(* Logix 5000 project; controller Comas_L4 vendor 1 type 14 code 193 rev 30.11; software revision 30.02; part 9 of 12 *)
(* tags used below, declared in another part *)
   Activation_Mode_Once : BOOL;
   Activation_Pompe : BOOL;
   Activation_Synchro_Directe_Codeur : BOOL;
   AOI_Pilotage_Codeur_Vitesse_Moy : Pilotage_Vitesse_Rapide_V4;
   Axe_Comas : MOTION_GROUP;
   Axe_Coupe_Fil : AXIS_CIP_DRIVE;
   Axe_Horizontal_Droit : AXIS_CIP_DRIVE;
   Axe_Horizontal_Gauche : AXIS_CIP_DRIVE;
   Axe_Pompe_Doseuse : AXIS_CIP_DRIVE;
   Axe_Vertical_Droit : AXIS_CIP_DRIVE;
   Axe_Vertical_Gauche : AXIS_CIP_DRIVE;
   Axe_Virtuel_Codeur : AXIS_VIRTUAL;
   Axe_Virtuel_Maitre : AXIS_VIRTUAL;
   CAM_Inter_Virtuel_Maitre : CAM[100];
   CamGenerator_Horizontal : AOI_CamGenerator_ST;
   CamGenerator_Vertical : AOI_CamGenerator_ST;
   CO_Acquit_defaut : BOOL;
   CO_Activation : BOOL;
   CO_Axe_Reel_Desynchro : BOOL;
   CO_Axe_Reel_En_Synchro : BOOL;
   CO_Consigne_Pompe_Acc_Dec : REAL;
   CO_Consigne_Pompe_Jerk : REAL;
   CO_Control_Pompe_Vitesse : REAL;
   CO_Degagement_En_Cours : BOOL;
   CO_Degagement_Possible : BOOL;
   CO_demande_darret : BOOL;
   CO_Demande_Init : BOOL;
   CO_en_Marche : BOOL;
   CO_Engage_Axe_Coupe_Fil : Engage_Axe;
   CO_Engage_Axe_H_Droit : Engage_Axe;
   CO_Engage_Axe_H_Gauche : Engage_Axe;
   CO_Engage_Axe_V_Droit : Engage_Axe;
   CO_Engage_Axe_V_Gauche : Engage_Axe;
   CO_Engage_Maitre : Engage_Axe_Virtuel;
   CO_Engagement : BOOL;
   CO_Engagement_Maitre : BOOL;
   CO_Front_Demande_Init : BOOL;
   CO_Front_Raz_Init : BOOL;
   CO_Front_Reset_Init_OK : BOOL;
   CO_Init_Coupe_Fil : BOOL;
   CO_Init_Horizontal_Droit : BOOL;
   CO_Init_Horizontal_Gauche : BOOL;
   CO_Init_Ok : BOOL;
   CO_Init_Pompe_Doseuse : BOOL;
   CO_Init_Vertical_Droit : BOOL;
   CO_Init_Vertical_Gauche : BOOL;
   CO_Machine_sans_defaut : BOOL;
   CO_Synchro_Axe_En_Cours : BOOL;
   CO_Temp_Activation : TIMER;
   CO_Temp_Desynchro : TIMER;
   CO_Temp_Pret : TIMER;
   CO_Tempo_Demande_Init : TIMER;
   CO_Tempo_Engagement : TIMER;
   CO_TON_Activation : TIMER;
   CO_Top_Degagement : BOOL;
   CO_Top_Depart_Pompe_Avance : BOOL;
   CO_Top_Depart_Pompe_Inter1 : BOOL;
   CO_Top_Depart_Pompe_Inter2 : BOOL;
   CO_Top_Depart_Pompe_Inter3 : BOOL;
   CO_Top_Depart_Pompe_Inter4 : BOOL;
   CO_Top_Depart_Pompe_Inter5 : BOOL;
   CO_Top_Depart_Pompe_Inter6 : BOOL;
   CO_Top_Depart_Pompe_Inter7 : BOOL;
   CO_Top_Depart_Pompe_Inter8 : BOOL;
   CO_Top_Depart_Pompe_Recul : BOOL;
   CO_Top_Once_Axe_Virtuel : BOOL;
   Init_Coupe_Fil : Init_Axe_CIP;
   Init_Horizontal_Droit : Init_Axe_CIP;
   Init_Horizontal_Gauche : Init_Axe_CIP;
   Init_Pompe_Doseuse : Init_Axe_CIP;
   Init_Vertical_Droit : Init_Axe_CIP;
   Init_Vertical_Gauche : Init_Axe_CIP;
   Output_Cams_Degagement : Output_Cams;
   Output_Cams_Pompe_Avance : Output_Cams;
   Output_Cams_Pompe_Inter1 : Output_Cams;
   Output_Cams_Pompe_Inter2 : Output_Cams;
   Output_Cams_Pompe_Inter3 : Output_Cams;
   Output_Cams_Pompe_Inter4 : Output_Cams;
   Output_Cams_Pompe_Inter5 : Output_Cams;
   Output_Cams_Pompe_Inter6 : Output_Cams;
   Output_Cams_Pompe_Inter7 : Output_Cams;
   Output_Cams_Pompe_Inter8 : Output_Cams;
   Output_Cams_Pompe_Recul : Output_Cams;
   PCAM_Horizontal : UDT_CamGeneration;
   PCAM_Inter_PCAM_Horizontal : CAM[100];
   PCAM_Inter_PCAM_Vertical : CAM[100];
   PCAM_Vertical : UDT_CamGeneration;
   RECETTE_EC : UDT_RECIPE;
   RSW_CO_Demande_Initialisation : BOOL;
   RSW_Depose_Active : BOOL;
   Speed_Control_Pompe : Axis_speed_control;
   Tempo_RAZ_Ton_Once : TIMER;
   Vitesse_Moy_Codeur : REAL;
(* Comas, continued *)

ROUTINE E00_Initialisation   (* ladder *)
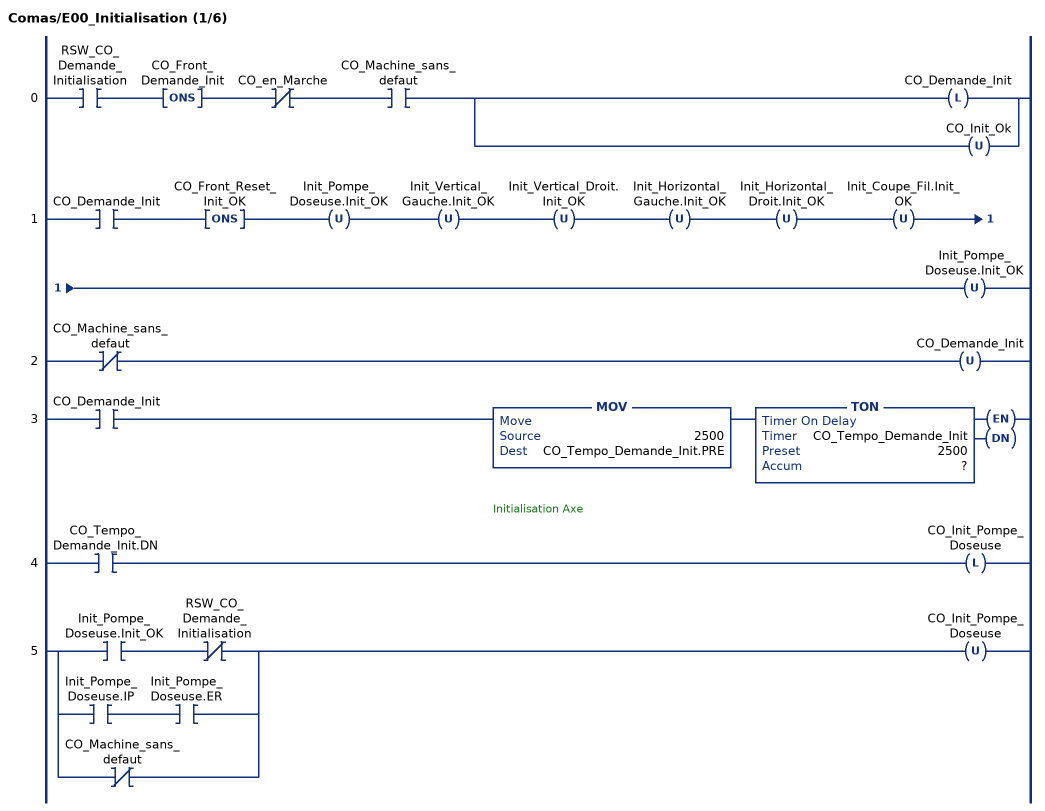
   0: XIC(RSW_CO_Demande_Initialisation)ONS(CO_Front_Demande_Init)XIO(CO_en_Marche)XIC(CO_Machine_sans_defaut)[OTL(CO_Demande_Init) ,OTU(CO_Init_Ok) ];
   1: XIC(CO_Demande_Init)ONS(CO_Front_Reset_Init_OK)OTU(Init_Pompe_Doseuse.Init_OK)OTU(Init_Vertical_Gauche.Init_OK)OTU(Init_Vertical_Droit.Init_OK)OTU(Init_Horizontal_Gauche.Init_OK)OTU(Init_Horizontal_Droit.Init_OK)OTU(Init_Coupe_Fil.Init_OK)OTU(Init_Pompe_Doseuse.Init_OK);
   2: XIO(CO_Machine_sans_defaut)OTU(CO_Demande_Init);
   3: XIC(CO_Demande_Init)MOV(2500,CO_Tempo_Demande_Init.PRE)TON(CO_Tempo_Demande_Init,?,?);
   // Initialisation Axe
   4: XIC(CO_Tempo_Demande_Init.DN)OTL(CO_Init_Pompe_Doseuse);
   5: [XIC(Init_Pompe_Doseuse.Init_OK) XIO(RSW_CO_Demande_Initialisation) ,XIC(Init_Pompe_Doseuse.IP) XIC(Init_Pompe_Doseuse.ER) ,XIO(CO_Machine_sans_defaut) ]OTU(CO_Init_Pompe_Doseuse);
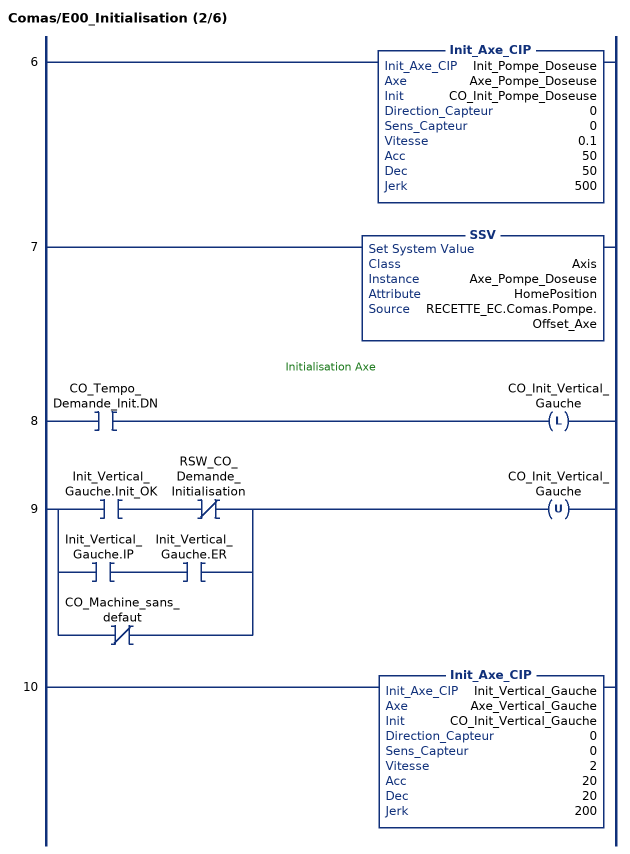
   6: Init_Axe_CIP(Init_Pompe_Doseuse,Axe_Pompe_Doseuse,CO_Init_Pompe_Doseuse,0,0,0.1,50,50,500);
   7: SSV(Axis,Axe_Pompe_Doseuse,HomePosition,RECETTE_EC.Comas.Pompe.Offset_Axe);
   // Initialisation Axe
   8: XIC(CO_Tempo_Demande_Init.DN)OTL(CO_Init_Vertical_Gauche);
   9: [XIC(Init_Vertical_Gauche.Init_OK) XIO(RSW_CO_Demande_Initialisation) ,XIC(Init_Vertical_Gauche.IP) XIC(Init_Vertical_Gauche.ER) ,XIO(CO_Machine_sans_defaut) ]OTU(CO_Init_Vertical_Gauche);
   10: Init_Axe_CIP(Init_Vertical_Gauche,Axe_Vertical_Gauche,CO_Init_Vertical_Gauche,0,0,2,20,20,200);
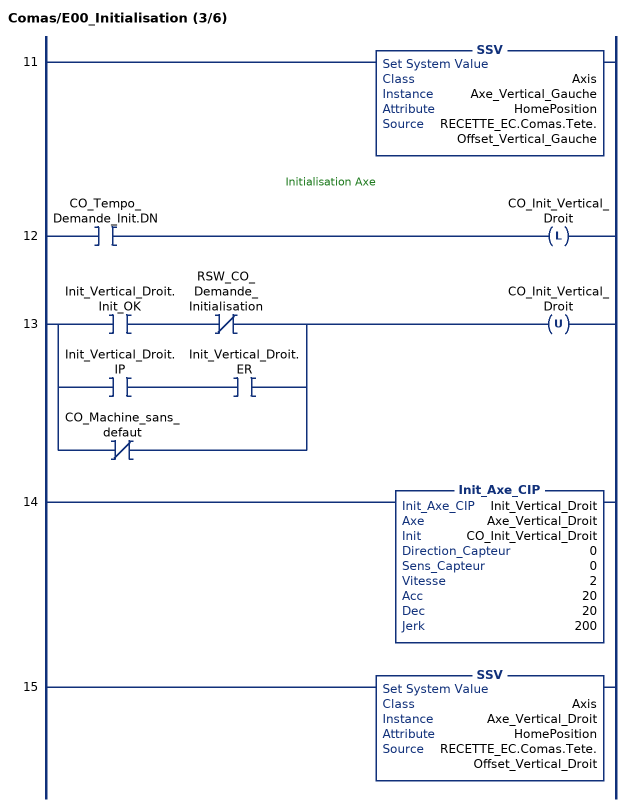
   11: SSV(Axis,Axe_Vertical_Gauche,HomePosition,RECETTE_EC.Comas.Tete.Offset_Vertical_Gauche);
   // Initialisation Axe
   12: XIC(CO_Tempo_Demande_Init.DN)OTL(CO_Init_Vertical_Droit);
   13: [XIC(Init_Vertical_Droit.Init_OK) XIO(RSW_CO_Demande_Initialisation) ,XIC(Init_Vertical_Droit.IP) XIC(Init_Vertical_Droit.ER) ,XIO(CO_Machine_sans_defaut) ]OTU(CO_Init_Vertical_Droit);
   14: Init_Axe_CIP(Init_Vertical_Droit,Axe_Vertical_Droit,CO_Init_Vertical_Droit,0,0,2,20,20,200);
   15: SSV(Axis,Axe_Vertical_Droit,HomePosition,RECETTE_EC.Comas.Tete.Offset_Vertical_Droit);
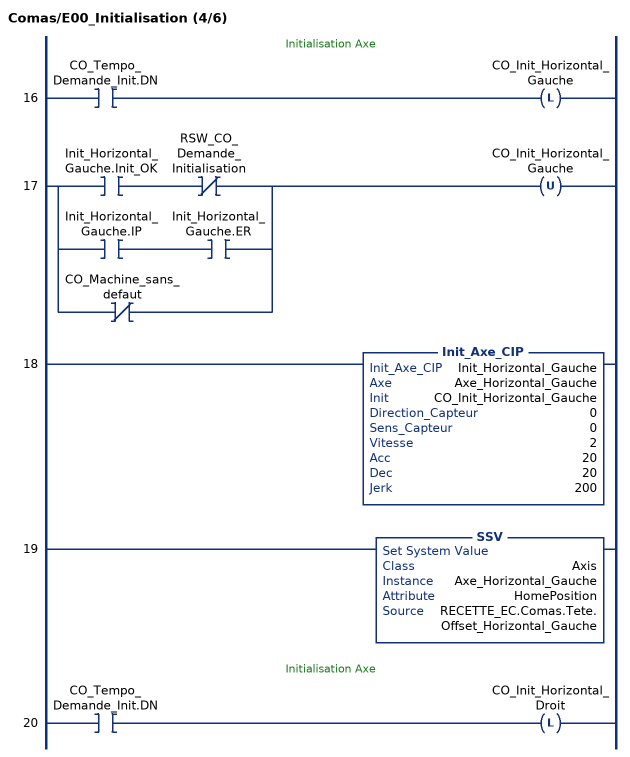
   // Initialisation Axe
   16: XIC(CO_Tempo_Demande_Init.DN)OTL(CO_Init_Horizontal_Gauche);
   17: [XIC(Init_Horizontal_Gauche.Init_OK) XIO(RSW_CO_Demande_Initialisation) ,XIC(Init_Horizontal_Gauche.IP) XIC(Init_Horizontal_Gauche.ER) ,XIO(CO_Machine_sans_defaut) ]OTU(CO_Init_Horizontal_Gauche);
   18: Init_Axe_CIP(Init_Horizontal_Gauche,Axe_Horizontal_Gauche,CO_Init_Horizontal_Gauche,0,0,2,20,20,200);
   19: SSV(Axis,Axe_Horizontal_Gauche,HomePosition,RECETTE_EC.Comas.Tete.Offset_Horizontal_Gauche);
   // Initialisation Axe
   20: XIC(CO_Tempo_Demande_Init.DN)OTL(CO_Init_Horizontal_Droit);
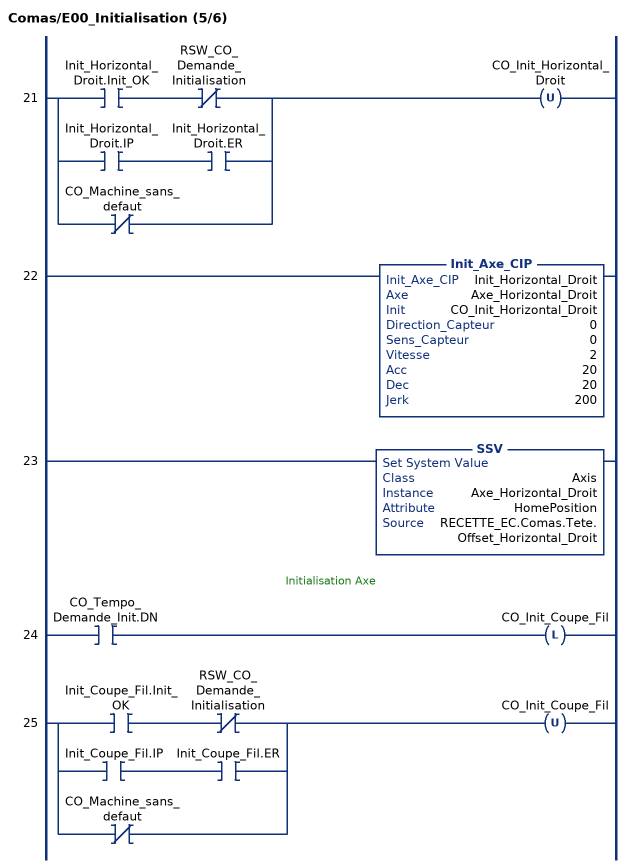
   21: [XIC(Init_Horizontal_Droit.Init_OK) XIO(RSW_CO_Demande_Initialisation) ,XIC(Init_Horizontal_Droit.IP) XIC(Init_Horizontal_Droit.ER) ,XIO(CO_Machine_sans_defaut) ]OTU(CO_Init_Horizontal_Droit);
   22: Init_Axe_CIP(Init_Horizontal_Droit,Axe_Horizontal_Droit,CO_Init_Horizontal_Droit,0,0,2,20,20,200);
   23: SSV(Axis,Axe_Horizontal_Droit,HomePosition,RECETTE_EC.Comas.Tete.Offset_Horizontal_Droit);
   // Initialisation Axe
   24: XIC(CO_Tempo_Demande_Init.DN)OTL(CO_Init_Coupe_Fil);
   25: [XIC(Init_Coupe_Fil.Init_OK) XIO(RSW_CO_Demande_Initialisation) ,XIC(Init_Coupe_Fil.IP) XIC(Init_Coupe_Fil.ER) ,XIO(CO_Machine_sans_defaut) ]OTU(CO_Init_Coupe_Fil);
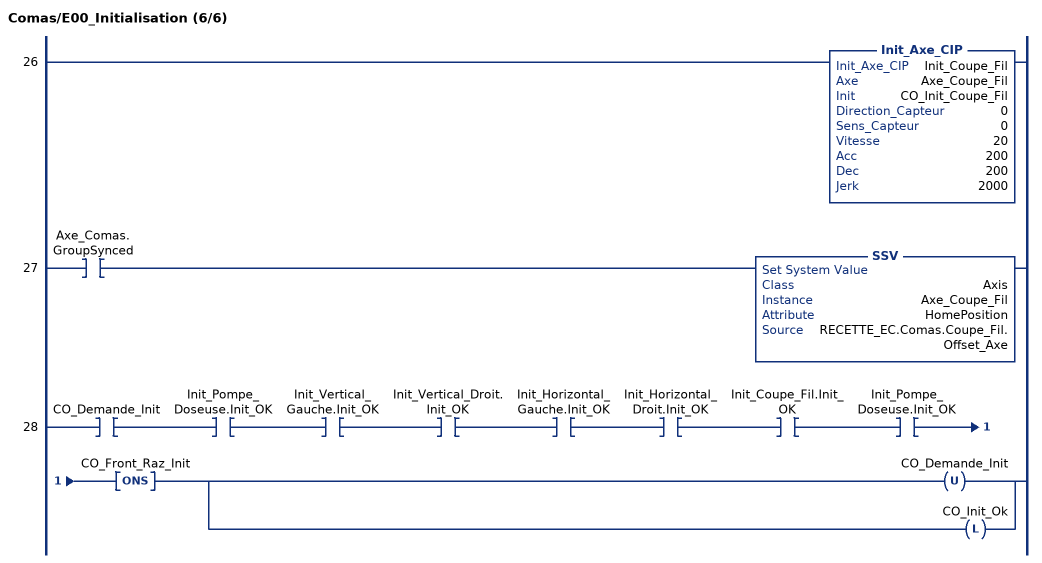
   26: Init_Axe_CIP(Init_Coupe_Fil,Axe_Coupe_Fil,CO_Init_Coupe_Fil,0,0,20,200,200,2000);
   27: XIC(Axe_Comas.GroupSynced)SSV(Axis,Axe_Coupe_Fil,HomePosition,RECETTE_EC.Comas.Coupe_Fil.Offset_Axe);
   28: XIC(CO_Demande_Init)XIC(Init_Pompe_Doseuse.Init_OK)XIC(Init_Vertical_Gauche.Init_OK)XIC(Init_Vertical_Droit.Init_OK)XIC(Init_Horizontal_Gauche.Init_OK)XIC(Init_Horizontal_Droit.Init_OK)XIC(Init_Coupe_Fil.Init_OK)XIC(Init_Pompe_Doseuse.Init_OK)ONS(CO_Front_Raz_Init)[OTU(CO_Demande_Init) ,OTL(CO_Init_Ok) ];
END_ROUTINE

ROUTINE F00_Engagement_Tete   (* ladder *)
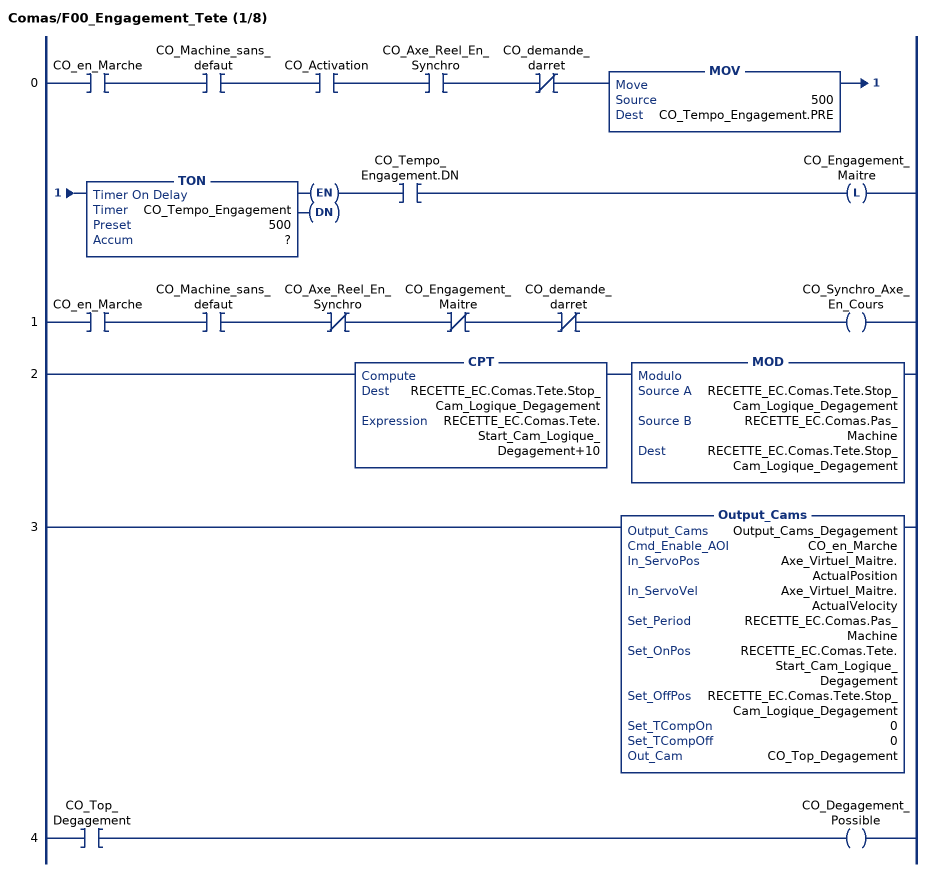
   0: XIC(CO_en_Marche)XIC(CO_Machine_sans_defaut)XIC(CO_Activation)XIC(CO_Axe_Reel_En_Synchro)XIO(CO_demande_darret)MOV(500,CO_Tempo_Engagement.PRE)TON(CO_Tempo_Engagement,?,?)XIC(CO_Tempo_Engagement.DN)OTL(CO_Engagement_Maitre);
   1: XIC(CO_en_Marche)XIC(CO_Machine_sans_defaut)XIO(CO_Axe_Reel_En_Synchro)XIO(CO_Engagement_Maitre)XIO(CO_demande_darret)OTE(CO_Synchro_Axe_En_Cours);
   2: CPT(RECETTE_EC.Comas.Tete.Stop_Cam_Logique_Degagement,RECETTE_EC.Comas.Tete.Start_Cam_Logique_Degagement+10)MOD(RECETTE_EC.Comas.Tete.Stop_Cam_Logique_Degagement,RECETTE_EC.Comas.Pas_Machine,RECETTE_EC.Comas.Tete.Stop_Cam_Logique_Degagement);
   3: Output_Cams(Output_Cams_Degagement,CO_en_Marche,Axe_Virtuel_Maitre.ActualPosition,Axe_Virtuel_Maitre.ActualVelocity,RECETTE_EC.Comas.Pas_Machine,RECETTE_EC.Comas.Tete.Start_Cam_Logique_Degagement,RECETTE_EC.Comas.Tete.Stop_Cam_Logique_Degagement,0,0,CO_Top_Degagement);
   4: XIC(CO_Top_Degagement)OTE(CO_Degagement_Possible);
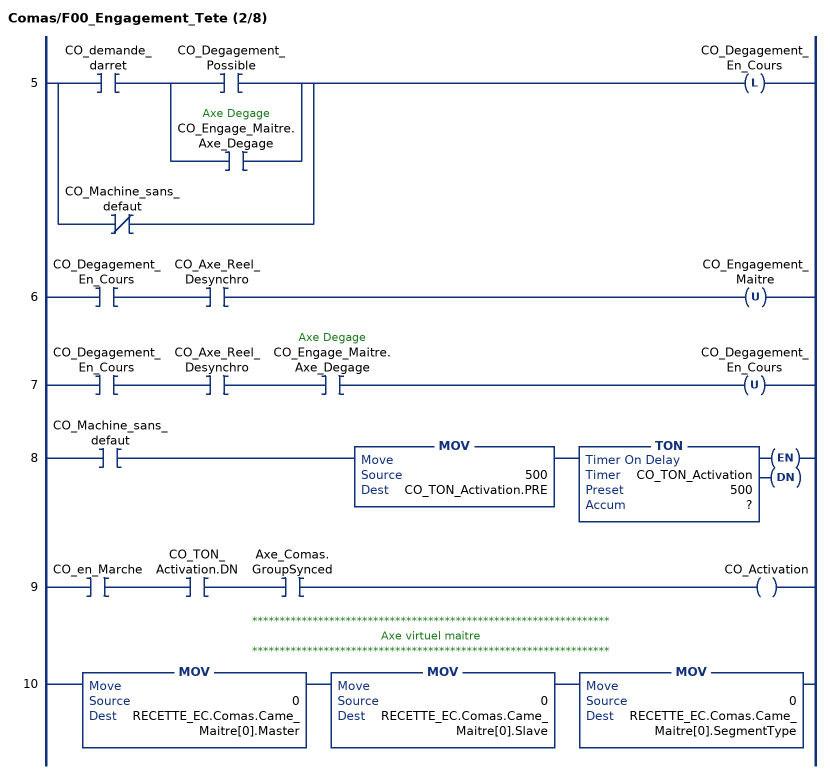
   5: [XIC(CO_demande_darret) [XIC(CO_Degagement_Possible) ,XIC(CO_Engage_Maitre.Axe_Degage) ] ,XIO(CO_Machine_sans_defaut) ]OTL(CO_Degagement_En_Cours);
   6: XIC(CO_Degagement_En_Cours)XIC(CO_Axe_Reel_Desynchro)OTU(CO_Engagement_Maitre);
   7: XIC(CO_Degagement_En_Cours)XIC(CO_Axe_Reel_Desynchro)XIC(CO_Engage_Maitre.Axe_Degage)OTU(CO_Degagement_En_Cours);
   8: XIC(CO_Machine_sans_defaut)MOV(500,CO_TON_Activation.PRE)TON(CO_TON_Activation,?,?);
   9: XIC(CO_en_Marche)XIC(CO_TON_Activation.DN)XIC(Axe_Comas.GroupSynced)OTE(CO_Activation);
   // *****************************************************************
   // Axe virtuel maitre
   // *****************************************************************
   10: MOV(0,RECETTE_EC.Comas.Came_Maitre[0].Master)MOV(0,RECETTE_EC.Comas.Came_Maitre[0].Slave)MOV(0,RECETTE_EC.Comas.Came_Maitre[0].SegmentType);
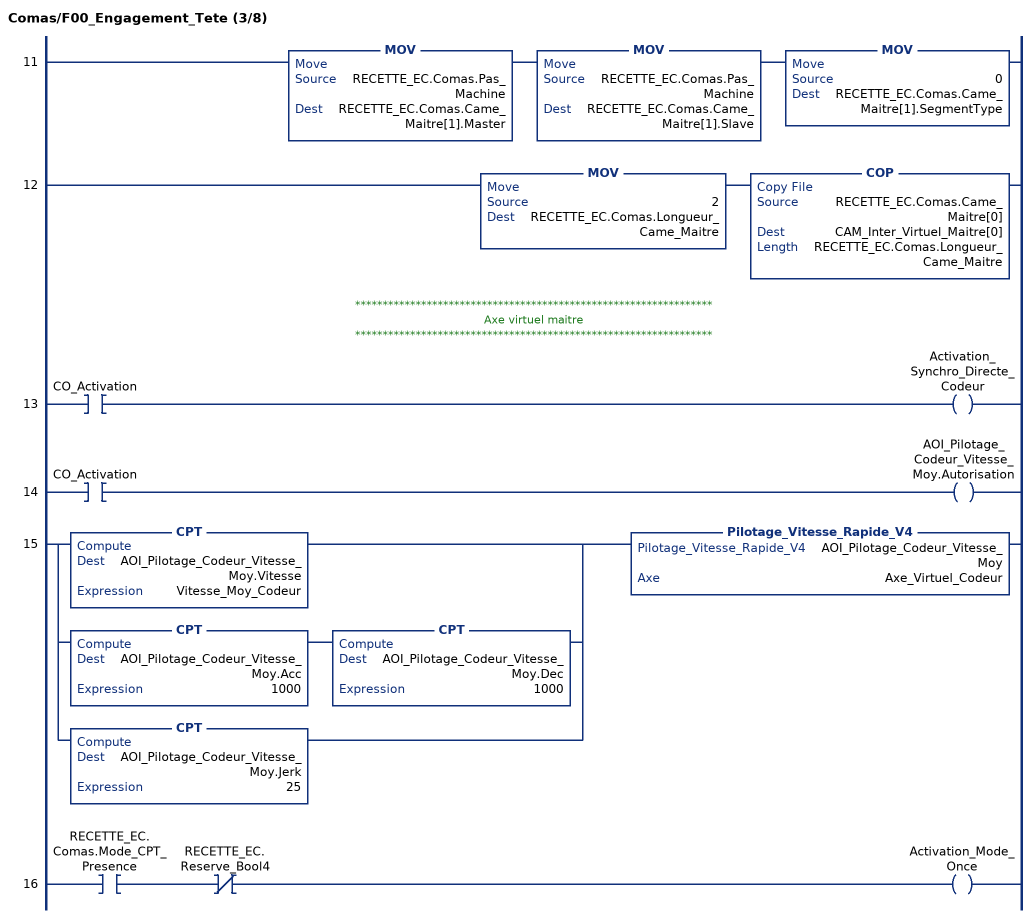
   11: MOV(RECETTE_EC.Comas.Pas_Machine,RECETTE_EC.Comas.Came_Maitre[1].Master)MOV(RECETTE_EC.Comas.Pas_Machine,RECETTE_EC.Comas.Came_Maitre[1].Slave)MOV(0,RECETTE_EC.Comas.Came_Maitre[1].SegmentType);
   12: MOV(2,RECETTE_EC.Comas.Longueur_Came_Maitre)COP(RECETTE_EC.Comas.Came_Maitre[0],CAM_Inter_Virtuel_Maitre[0],RECETTE_EC.Comas.Longueur_Came_Maitre);
   // *****************************************************************
   // Axe virtuel maitre
   // *****************************************************************
   13: XIC(CO_Activation)OTE(Activation_Synchro_Directe_Codeur);
   14: XIC(CO_Activation)OTE(AOI_Pilotage_Codeur_Vitesse_Moy.Autorisation);
   15: [CPT(AOI_Pilotage_Codeur_Vitesse_Moy.Vitesse,Vitesse_Moy_Codeur) ,CPT(AOI_Pilotage_Codeur_Vitesse_Moy.Acc,1000) CPT(AOI_Pilotage_Codeur_Vitesse_Moy.Dec,1000) ,CPT(AOI_Pilotage_Codeur_Vitesse_Moy.Jerk,25) ]Pilotage_Vitesse_Rapide_V4(AOI_Pilotage_Codeur_Vitesse_Moy,Axe_Virtuel_Codeur);
   16: XIC(RECETTE_EC.Comas.Mode_CPT_Presence)XIO(RECETTE_EC.Reserve_Bool4)OTE(Activation_Mode_Once);
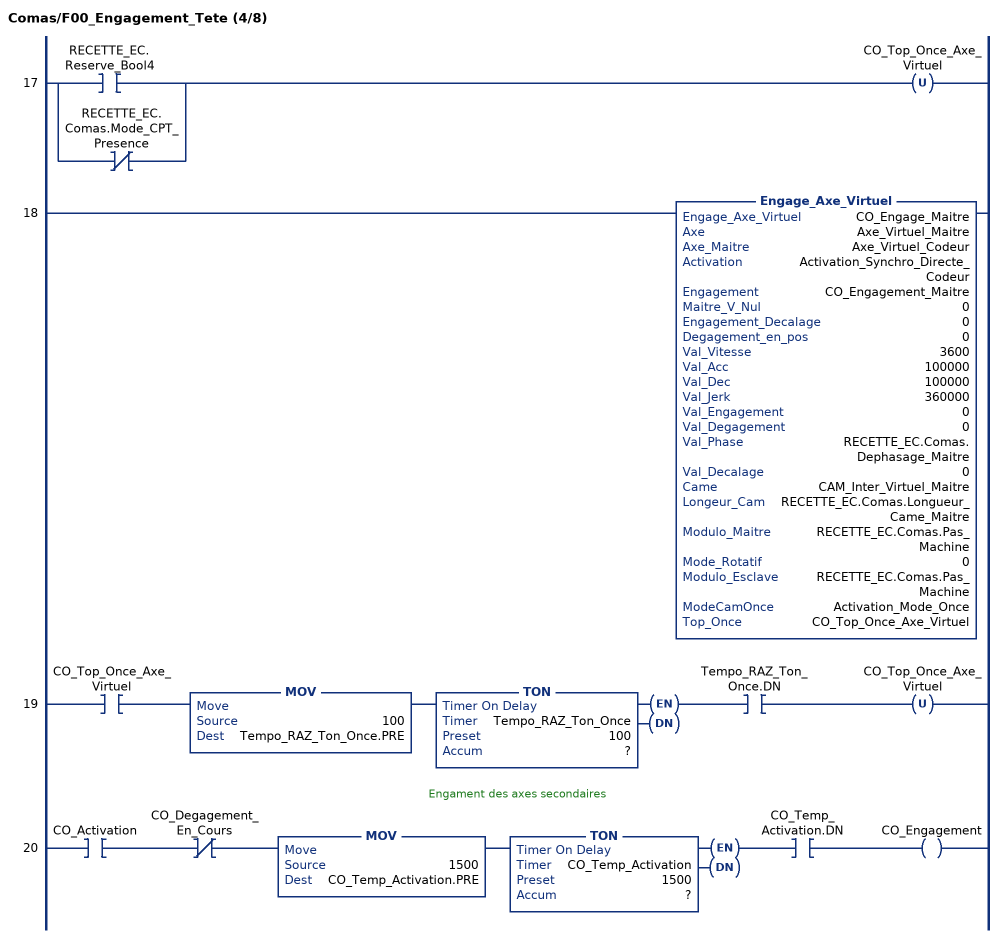
   17: [XIC(RECETTE_EC.Reserve_Bool4) ,XIO(RECETTE_EC.Comas.Mode_CPT_Presence) ]OTU(CO_Top_Once_Axe_Virtuel);
   18: Engage_Axe_Virtuel(CO_Engage_Maitre,Axe_Virtuel_Maitre,Axe_Virtuel_Codeur,Activation_Synchro_Directe_Codeur,CO_Engagement_Maitre,0,0,0,3600,100000,100000,360000,0,0,RECETTE_EC.Comas.Dephasage_Maitre,0,CAM_Inter_Virtuel_Maitre,RECETTE_EC.Comas.Longueur_Came_Maitre,RECETTE_EC.Comas.Pas_Machine,0,RECETTE_EC.Comas.Pas_Machine,Activation_Mode_Once,CO_Top_Once_Axe_Virtuel);
   19: XIC(CO_Top_Once_Axe_Virtuel)MOV(100,Tempo_RAZ_Ton_Once.PRE)TON(Tempo_RAZ_Ton_Once,?,?)XIC(Tempo_RAZ_Ton_Once.DN)OTU(CO_Top_Once_Axe_Virtuel);
   // Engament des axes secondaires
   20: XIC(CO_Activation)XIO(CO_Degagement_En_Cours)MOV(1500,CO_Temp_Activation.PRE)TON(CO_Temp_Activation,?,?)XIC(CO_Temp_Activation.DN)OTE(CO_Engagement);
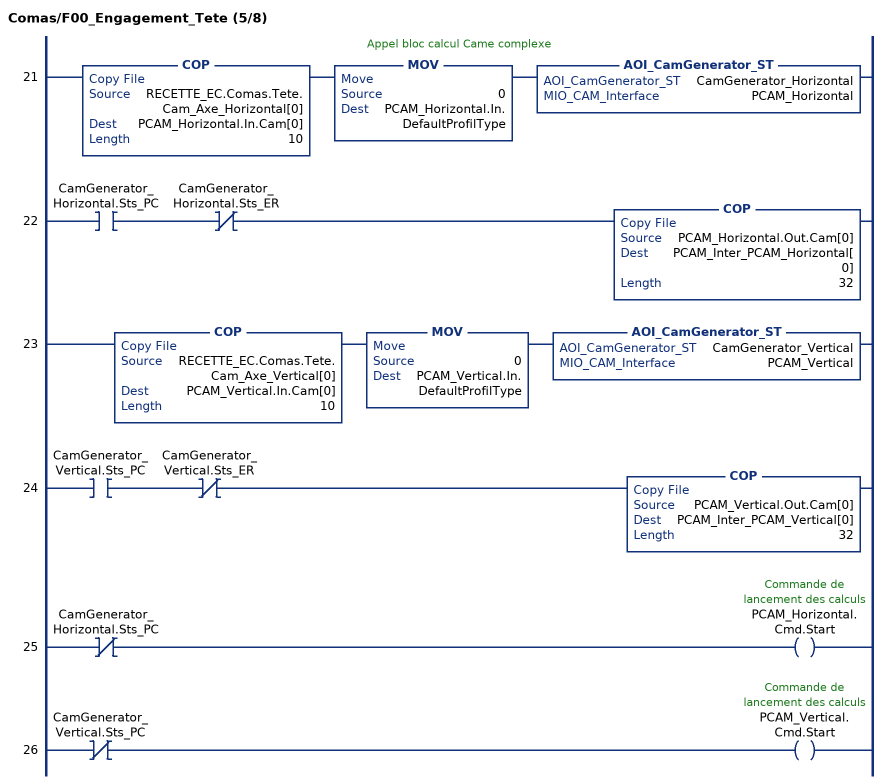
   // Appel bloc calcul Came complexe
   21: COP(RECETTE_EC.Comas.Tete.Cam_Axe_Horizontal[0],PCAM_Horizontal.In.Cam[0],10)MOV(0,PCAM_Horizontal.In.DefaultProfilType)AOI_CamGenerator_ST(CamGenerator_Horizontal,PCAM_Horizontal);
   22: XIC(CamGenerator_Horizontal.Sts_PC)XIO(CamGenerator_Horizontal.Sts_ER)COP(PCAM_Horizontal.Out.Cam[0],PCAM_Inter_PCAM_Horizontal[0],32);
   23: COP(RECETTE_EC.Comas.Tete.Cam_Axe_Vertical[0],PCAM_Vertical.In.Cam[0],10)MOV(0,PCAM_Vertical.In.DefaultProfilType)AOI_CamGenerator_ST(CamGenerator_Vertical,PCAM_Vertical);
   24: XIC(CamGenerator_Vertical.Sts_PC)XIO(CamGenerator_Vertical.Sts_ER)COP(PCAM_Vertical.Out.Cam[0],PCAM_Inter_PCAM_Vertical[0],32);
   25: XIO(CamGenerator_Horizontal.Sts_PC)OTE(PCAM_Horizontal.Cmd.Start);
   26: XIO(CamGenerator_Vertical.Sts_PC)OTE(PCAM_Vertical.Cmd.Start);
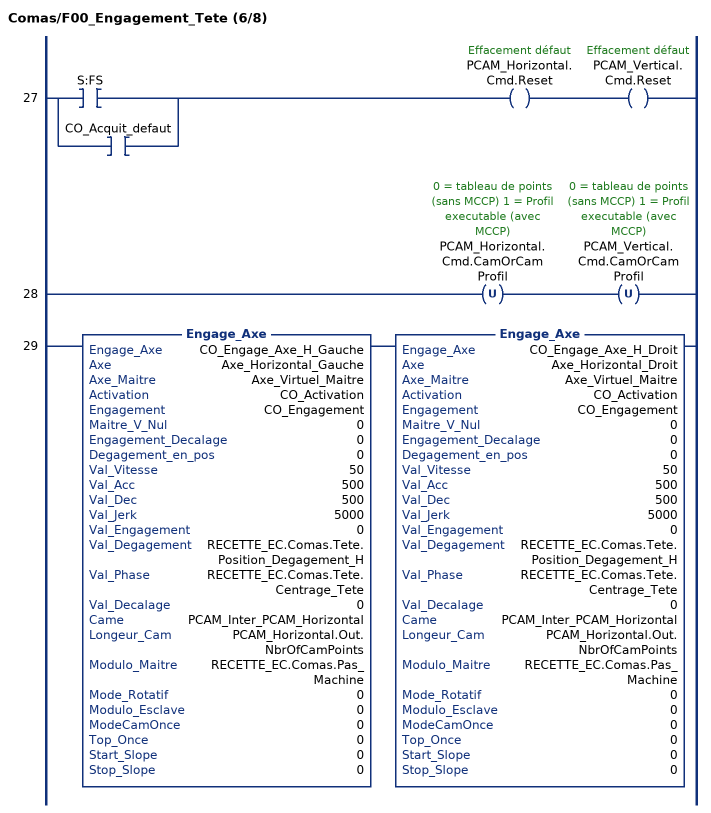
   27: [XIC(S:FS) ,XIC(CO_Acquit_defaut) ]OTE(PCAM_Horizontal.Cmd.Reset)OTE(PCAM_Vertical.Cmd.Reset);
   28: OTU(PCAM_Horizontal.Cmd.CamOrCamProfil)OTU(PCAM_Vertical.Cmd.CamOrCamProfil);
   29: Engage_Axe(CO_Engage_Axe_H_Gauche,Axe_Horizontal_Gauche,Axe_Virtuel_Maitre,CO_Activation,CO_Engagement,0,0,0,50,500,500,5000,0,RECETTE_EC.Comas.Tete.Position_Degagement_H,RECETTE_EC.Comas.Tete.Centrage_Tete,0,PCAM_Inter_PCAM_Horizontal,PCAM_Horizontal.Out.NbrOfCamPoints,RECETTE_EC.Comas.Pas_Machine,0,0,0,0,0,0)Engage_Axe(CO_Engage_Axe_H_Droit,Axe_Horizontal_Droit,Axe_Virtuel_Maitre,CO_Activation,CO_Engagement,0,0,0,50,500,500,5000,0,RECETTE_EC.Comas.Tete.Position_Degagement_H,RECETTE_EC.Comas.Tete.Centrage_Tete,0,PCAM_Inter_PCAM_Horizontal,PCAM_Horizontal.Out.NbrOfCamPoints,RECETTE_EC.Comas.Pas_Machine,0,0,0,0,0,0);
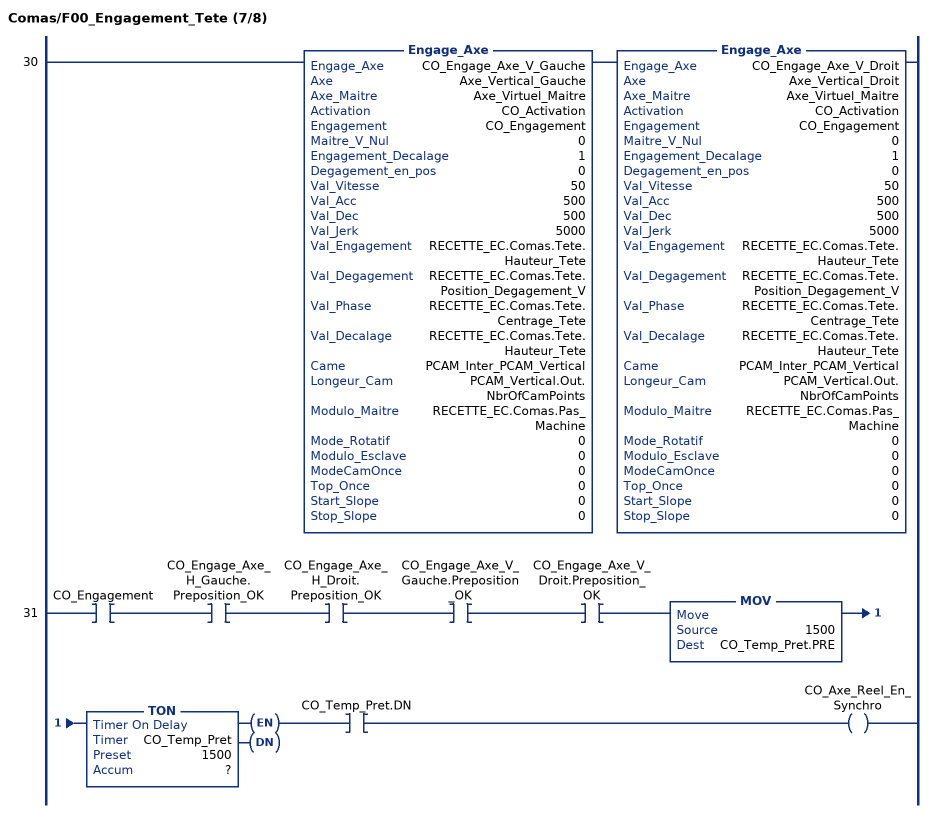
   30: Engage_Axe(CO_Engage_Axe_V_Gauche,Axe_Vertical_Gauche,Axe_Virtuel_Maitre,CO_Activation,CO_Engagement,0,1,0,50,500,500,5000,RECETTE_EC.Comas.Tete.Hauteur_Tete,RECETTE_EC.Comas.Tete.Position_Degagement_V,RECETTE_EC.Comas.Tete.Centrage_Tete,RECETTE_EC.Comas.Tete.Hauteur_Tete,PCAM_Inter_PCAM_Vertical,PCAM_Vertical.Out.NbrOfCamPoints,RECETTE_EC.Comas.Pas_Machine,0,0,0,0,0,0)Engage_Axe(CO_Engage_Axe_V_Droit,Axe_Vertical_Droit,Axe_Virtuel_Maitre,CO_Activation,CO_Engagement,0,1,0,50,500,500,5000,RECETTE_EC.Comas.Tete.Hauteur_Tete,RECETTE_EC.Comas.Tete.Position_Degagement_V,RECETTE_EC.Comas.Tete.Centrage_Tete,RECETTE_EC.Comas.Tete.Hauteur_Tete,PCAM_Inter_PCAM_Vertical,PCAM_Vertical.Out.NbrOfCamPoints,RECETTE_EC.Comas.Pas_Machine,0,0,0,0,0,0);
   31: XIC(CO_Engagement)XIC(CO_Engage_Axe_H_Gauche.Preposition_OK)XIC(CO_Engage_Axe_H_Droit.Preposition_OK)XIC(CO_Engage_Axe_V_Gauche.Preposition_OK)XIC(CO_Engage_Axe_V_Droit.Preposition_OK)MOV(1500,CO_Temp_Pret.PRE)TON(CO_Temp_Pret,?,?)XIC(CO_Temp_Pret.DN)OTE(CO_Axe_Reel_En_Synchro);
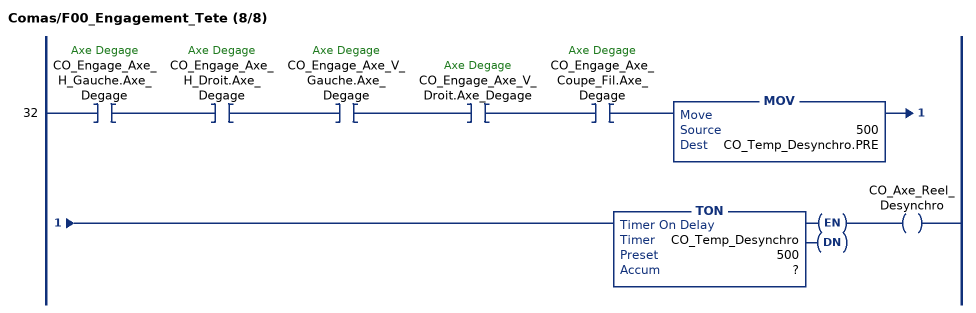
   32: XIC(CO_Engage_Axe_H_Gauche.Axe_Degage)XIC(CO_Engage_Axe_H_Droit.Axe_Degage)XIC(CO_Engage_Axe_V_Gauche.Axe_Degage)XIC(CO_Engage_Axe_V_Droit.Axe_Degage)XIC(CO_Engage_Axe_Coupe_Fil.Axe_Degage)MOV(500,CO_Temp_Desynchro.PRE)TON(CO_Temp_Desynchro,?,?)OTE(CO_Axe_Reel_Desynchro);
END_ROUTINE

ROUTINE F01_Engagement_Pompe   (* ladder *)
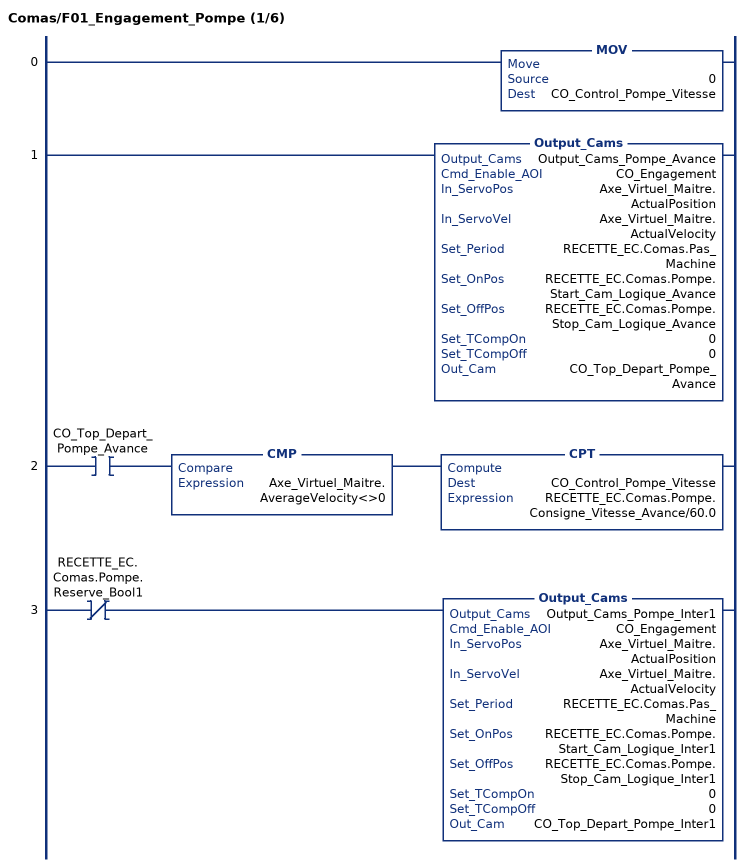
   0: MOV(0,CO_Control_Pompe_Vitesse);
   1: Output_Cams(Output_Cams_Pompe_Avance,CO_Engagement,Axe_Virtuel_Maitre.ActualPosition,Axe_Virtuel_Maitre.ActualVelocity,RECETTE_EC.Comas.Pas_Machine,RECETTE_EC.Comas.Pompe.Start_Cam_Logique_Avance,RECETTE_EC.Comas.Pompe.Stop_Cam_Logique_Avance,0,0,CO_Top_Depart_Pompe_Avance);
   2: XIC(CO_Top_Depart_Pompe_Avance)CMP(Axe_Virtuel_Maitre.AverageVelocity<>0)CPT(CO_Control_Pompe_Vitesse,RECETTE_EC.Comas.Pompe.Consigne_Vitesse_Avance/60.0);
   3: XIO(RECETTE_EC.Comas.Pompe.Reserve_Bool1)Output_Cams(Output_Cams_Pompe_Inter1,CO_Engagement,Axe_Virtuel_Maitre.ActualPosition,Axe_Virtuel_Maitre.ActualVelocity,RECETTE_EC.Comas.Pas_Machine,RECETTE_EC.Comas.Pompe.Start_Cam_Logique_Inter1,RECETTE_EC.Comas.Pompe.Stop_Cam_Logique_Inter1,0,0,CO_Top_Depart_Pompe_Inter1);
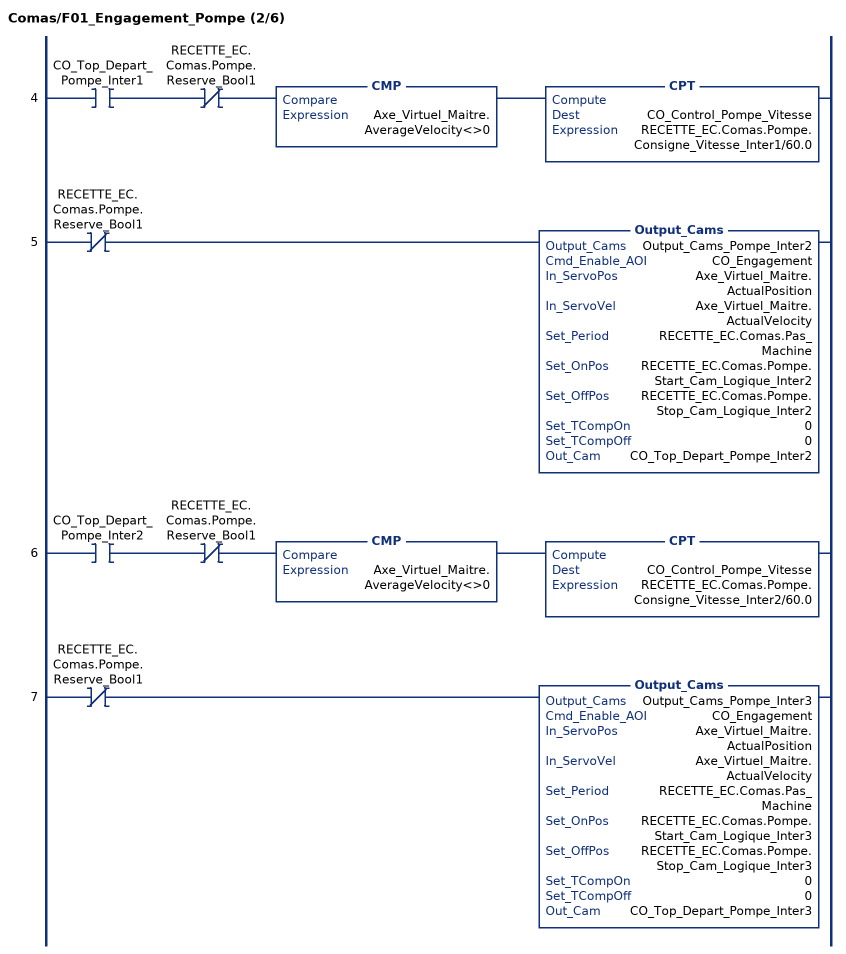
   4: XIC(CO_Top_Depart_Pompe_Inter1)XIO(RECETTE_EC.Comas.Pompe.Reserve_Bool1)CMP(Axe_Virtuel_Maitre.AverageVelocity<>0)CPT(CO_Control_Pompe_Vitesse,RECETTE_EC.Comas.Pompe.Consigne_Vitesse_Inter1/60.0);
   5: XIO(RECETTE_EC.Comas.Pompe.Reserve_Bool1)Output_Cams(Output_Cams_Pompe_Inter2,CO_Engagement,Axe_Virtuel_Maitre.ActualPosition,Axe_Virtuel_Maitre.ActualVelocity,RECETTE_EC.Comas.Pas_Machine,RECETTE_EC.Comas.Pompe.Start_Cam_Logique_Inter2,RECETTE_EC.Comas.Pompe.Stop_Cam_Logique_Inter2,0,0,CO_Top_Depart_Pompe_Inter2);
   6: XIC(CO_Top_Depart_Pompe_Inter2)XIO(RECETTE_EC.Comas.Pompe.Reserve_Bool1)CMP(Axe_Virtuel_Maitre.AverageVelocity<>0)CPT(CO_Control_Pompe_Vitesse,RECETTE_EC.Comas.Pompe.Consigne_Vitesse_Inter2/60.0);
   7: XIO(RECETTE_EC.Comas.Pompe.Reserve_Bool1)Output_Cams(Output_Cams_Pompe_Inter3,CO_Engagement,Axe_Virtuel_Maitre.ActualPosition,Axe_Virtuel_Maitre.ActualVelocity,RECETTE_EC.Comas.Pas_Machine,RECETTE_EC.Comas.Pompe.Start_Cam_Logique_Inter3,RECETTE_EC.Comas.Pompe.Stop_Cam_Logique_Inter3,0,0,CO_Top_Depart_Pompe_Inter3);
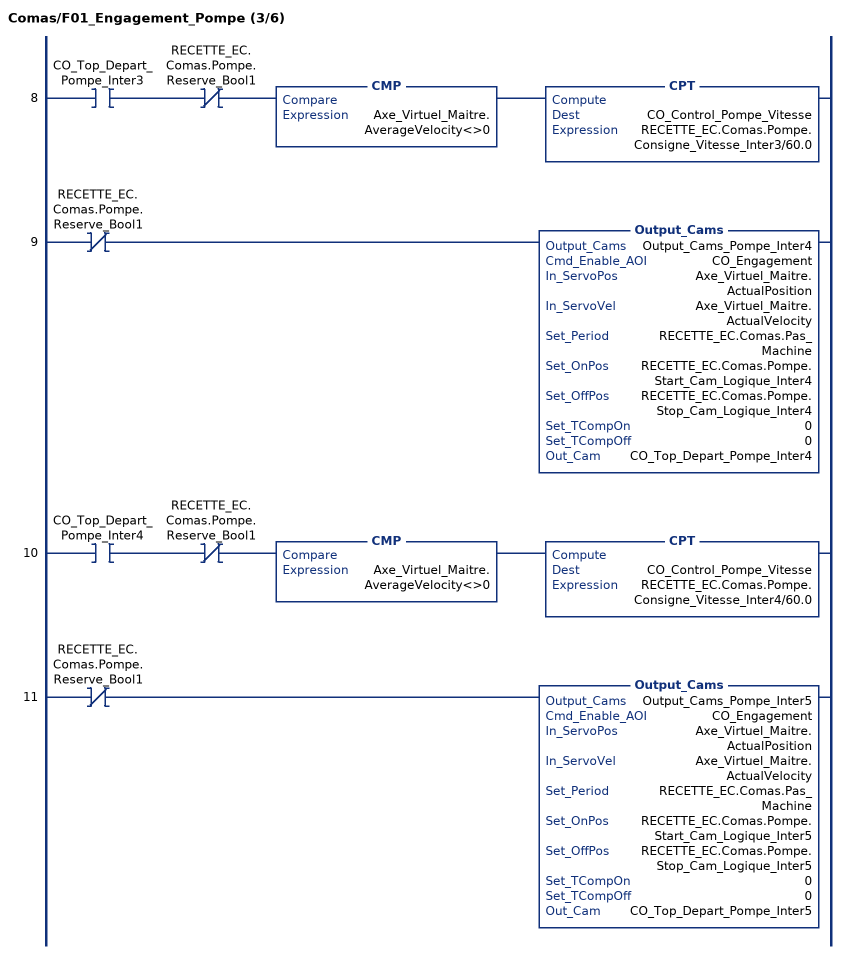
   8: XIC(CO_Top_Depart_Pompe_Inter3)XIO(RECETTE_EC.Comas.Pompe.Reserve_Bool1)CMP(Axe_Virtuel_Maitre.AverageVelocity<>0)CPT(CO_Control_Pompe_Vitesse,RECETTE_EC.Comas.Pompe.Consigne_Vitesse_Inter3/60.0);
   9: XIO(RECETTE_EC.Comas.Pompe.Reserve_Bool1)Output_Cams(Output_Cams_Pompe_Inter4,CO_Engagement,Axe_Virtuel_Maitre.ActualPosition,Axe_Virtuel_Maitre.ActualVelocity,RECETTE_EC.Comas.Pas_Machine,RECETTE_EC.Comas.Pompe.Start_Cam_Logique_Inter4,RECETTE_EC.Comas.Pompe.Stop_Cam_Logique_Inter4,0,0,CO_Top_Depart_Pompe_Inter4);
   10: XIC(CO_Top_Depart_Pompe_Inter4)XIO(RECETTE_EC.Comas.Pompe.Reserve_Bool1)CMP(Axe_Virtuel_Maitre.AverageVelocity<>0)CPT(CO_Control_Pompe_Vitesse,RECETTE_EC.Comas.Pompe.Consigne_Vitesse_Inter4/60.0);
   11: XIO(RECETTE_EC.Comas.Pompe.Reserve_Bool1)Output_Cams(Output_Cams_Pompe_Inter5,CO_Engagement,Axe_Virtuel_Maitre.ActualPosition,Axe_Virtuel_Maitre.ActualVelocity,RECETTE_EC.Comas.Pas_Machine,RECETTE_EC.Comas.Pompe.Start_Cam_Logique_Inter5,RECETTE_EC.Comas.Pompe.Stop_Cam_Logique_Inter5,0,0,CO_Top_Depart_Pompe_Inter5);
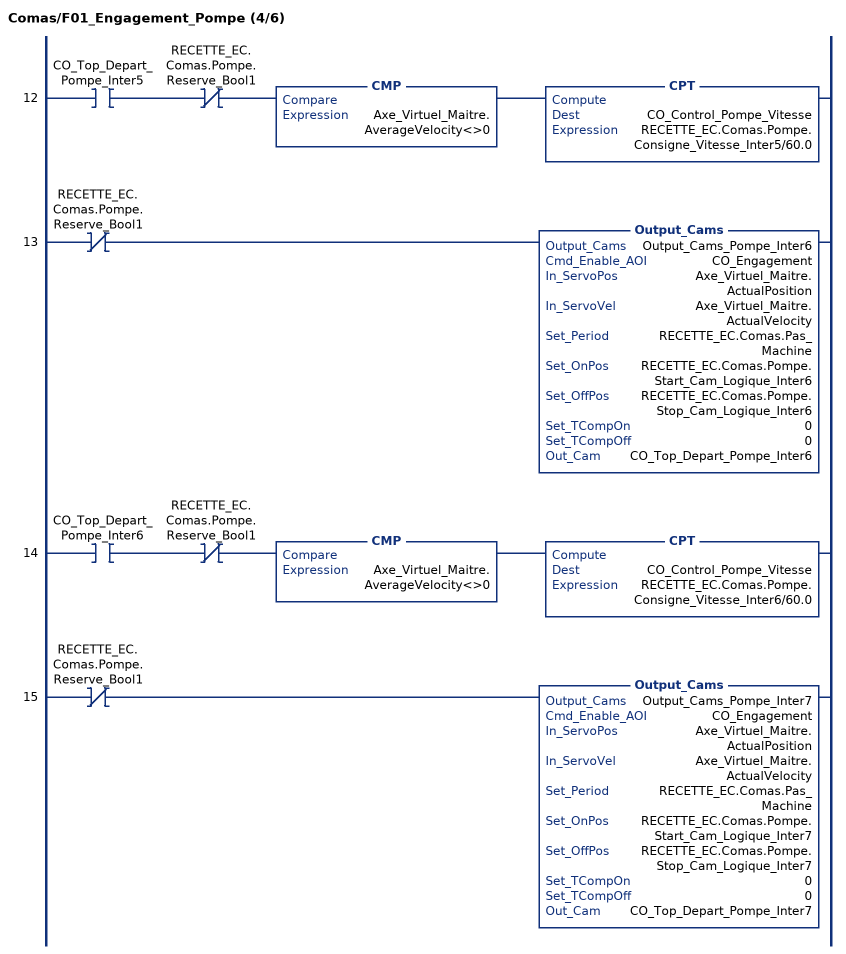
   12: XIC(CO_Top_Depart_Pompe_Inter5)XIO(RECETTE_EC.Comas.Pompe.Reserve_Bool1)CMP(Axe_Virtuel_Maitre.AverageVelocity<>0)CPT(CO_Control_Pompe_Vitesse,RECETTE_EC.Comas.Pompe.Consigne_Vitesse_Inter5/60.0);
   13: XIO(RECETTE_EC.Comas.Pompe.Reserve_Bool1)Output_Cams(Output_Cams_Pompe_Inter6,CO_Engagement,Axe_Virtuel_Maitre.ActualPosition,Axe_Virtuel_Maitre.ActualVelocity,RECETTE_EC.Comas.Pas_Machine,RECETTE_EC.Comas.Pompe.Start_Cam_Logique_Inter6,RECETTE_EC.Comas.Pompe.Stop_Cam_Logique_Inter6,0,0,CO_Top_Depart_Pompe_Inter6);
   14: XIC(CO_Top_Depart_Pompe_Inter6)XIO(RECETTE_EC.Comas.Pompe.Reserve_Bool1)CMP(Axe_Virtuel_Maitre.AverageVelocity<>0)CPT(CO_Control_Pompe_Vitesse,RECETTE_EC.Comas.Pompe.Consigne_Vitesse_Inter6/60.0);
   15: XIO(RECETTE_EC.Comas.Pompe.Reserve_Bool1)Output_Cams(Output_Cams_Pompe_Inter7,CO_Engagement,Axe_Virtuel_Maitre.ActualPosition,Axe_Virtuel_Maitre.ActualVelocity,RECETTE_EC.Comas.Pas_Machine,RECETTE_EC.Comas.Pompe.Start_Cam_Logique_Inter7,RECETTE_EC.Comas.Pompe.Stop_Cam_Logique_Inter7,0,0,CO_Top_Depart_Pompe_Inter7);
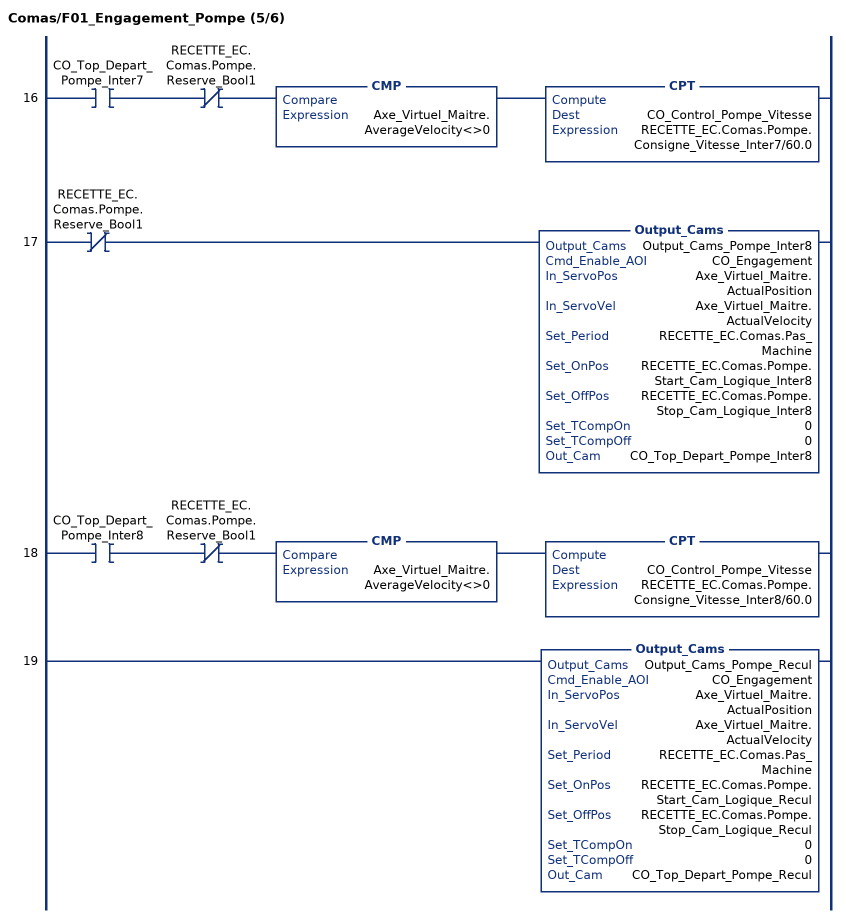
   16: XIC(CO_Top_Depart_Pompe_Inter7)XIO(RECETTE_EC.Comas.Pompe.Reserve_Bool1)CMP(Axe_Virtuel_Maitre.AverageVelocity<>0)CPT(CO_Control_Pompe_Vitesse,RECETTE_EC.Comas.Pompe.Consigne_Vitesse_Inter7/60.0);
   17: XIO(RECETTE_EC.Comas.Pompe.Reserve_Bool1)Output_Cams(Output_Cams_Pompe_Inter8,CO_Engagement,Axe_Virtuel_Maitre.ActualPosition,Axe_Virtuel_Maitre.ActualVelocity,RECETTE_EC.Comas.Pas_Machine,RECETTE_EC.Comas.Pompe.Start_Cam_Logique_Inter8,RECETTE_EC.Comas.Pompe.Stop_Cam_Logique_Inter8,0,0,CO_Top_Depart_Pompe_Inter8);
   18: XIC(CO_Top_Depart_Pompe_Inter8)XIO(RECETTE_EC.Comas.Pompe.Reserve_Bool1)CMP(Axe_Virtuel_Maitre.AverageVelocity<>0)CPT(CO_Control_Pompe_Vitesse,RECETTE_EC.Comas.Pompe.Consigne_Vitesse_Inter8/60.0);
   19: Output_Cams(Output_Cams_Pompe_Recul,CO_Engagement,Axe_Virtuel_Maitre.ActualPosition,Axe_Virtuel_Maitre.ActualVelocity,RECETTE_EC.Comas.Pas_Machine,RECETTE_EC.Comas.Pompe.Start_Cam_Logique_Recul,RECETTE_EC.Comas.Pompe.Stop_Cam_Logique_Recul,0,0,CO_Top_Depart_Pompe_Recul);
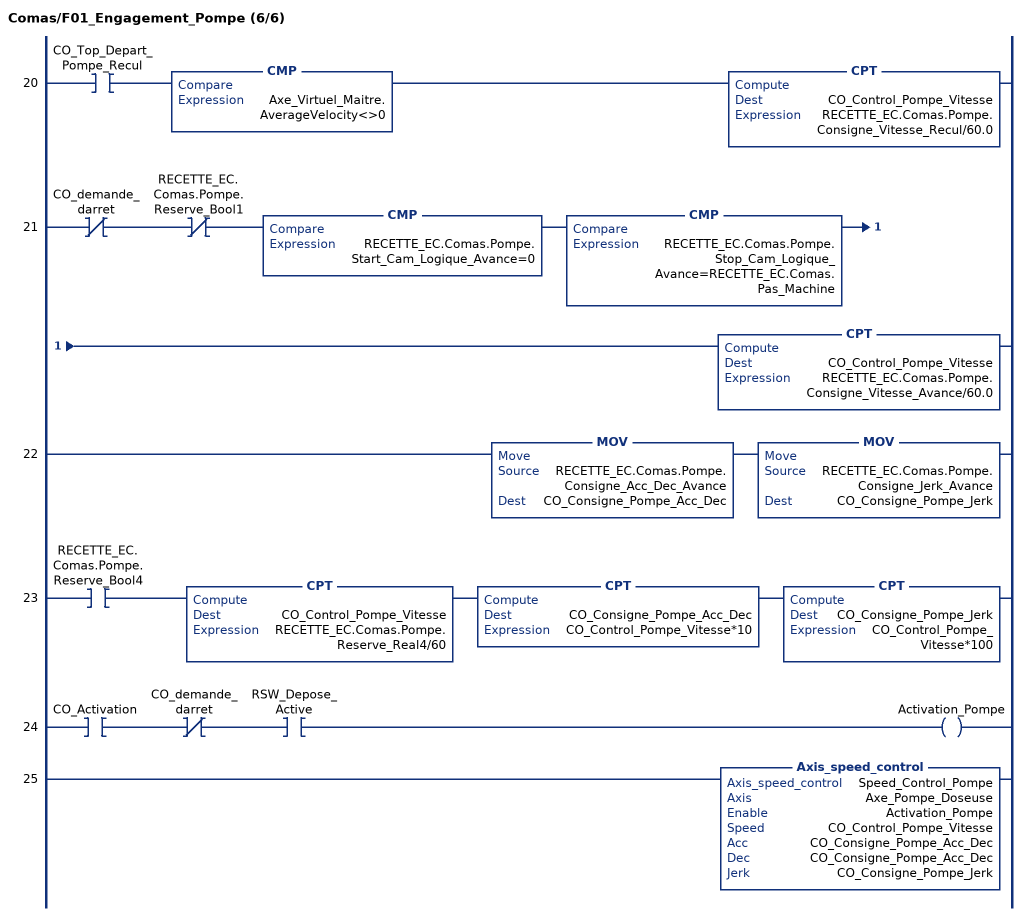
   20: XIC(CO_Top_Depart_Pompe_Recul)CMP(Axe_Virtuel_Maitre.AverageVelocity<>0)CPT(CO_Control_Pompe_Vitesse,RECETTE_EC.Comas.Pompe.Consigne_Vitesse_Recul/60.0);
   21: XIO(CO_demande_darret)XIO(RECETTE_EC.Comas.Pompe.Reserve_Bool1)CMP(RECETTE_EC.Comas.Pompe.Start_Cam_Logique_Avance=0)CMP(RECETTE_EC.Comas.Pompe.Stop_Cam_Logique_Avance=RECETTE_EC.Comas.Pas_Machine)CPT(CO_Control_Pompe_Vitesse,RECETTE_EC.Comas.Pompe.Consigne_Vitesse_Avance/60.0);
   22: MOV(RECETTE_EC.Comas.Pompe.Consigne_Acc_Dec_Avance,CO_Consigne_Pompe_Acc_Dec)MOV(RECETTE_EC.Comas.Pompe.Consigne_Jerk_Avance,CO_Consigne_Pompe_Jerk);
   23: XIC(RECETTE_EC.Comas.Pompe.Reserve_Bool4)CPT(CO_Control_Pompe_Vitesse,RECETTE_EC.Comas.Pompe.Reserve_Real4/60)CPT(CO_Consigne_Pompe_Acc_Dec,CO_Control_Pompe_Vitesse*10)CPT(CO_Consigne_Pompe_Jerk,CO_Control_Pompe_Vitesse*100);
   24: XIC(CO_Activation)XIO(CO_demande_darret)XIC(RSW_Depose_Active)OTE(Activation_Pompe);
   25: Axis_speed_control(Speed_Control_Pompe,Axe_Pompe_Doseuse,Activation_Pompe,CO_Control_Pompe_Vitesse,CO_Consigne_Pompe_Acc_Dec,CO_Consigne_Pompe_Acc_Dec,CO_Consigne_Pompe_Jerk);
END_ROUTINE
